% RSLogix 500 project ON DELAY.RSS, saved by version 8.30.00.16 %
PROJECT "UNTITLED"    % processor: MicroLogix 1000 %

PROGRAM FILES
  LAD 2 "MAIN_PROG"  4 rungs
  LAD 3 "START"  9 rungs
  LAD 4 "BUZZER"  7 rungs
  LAD 5 "STI_INT"  1 rungs
  LAD 6, 7, 8, 9, 10, 11, 12, 13, 14, 15, 16: only END

DATA FILES
  O0 OUTPUT  1 elements
  I1 INPUT  2 elements
  S2 STATUS  33 elements
  B3 BINARY  32 elements
  T4 TIMER  40 elements
  C5 COUNTER  32 elements
  R6 CONTROL  16 elements
  N7 INTEGER  105 elements

LADDER 2 "MAIN_PROG"
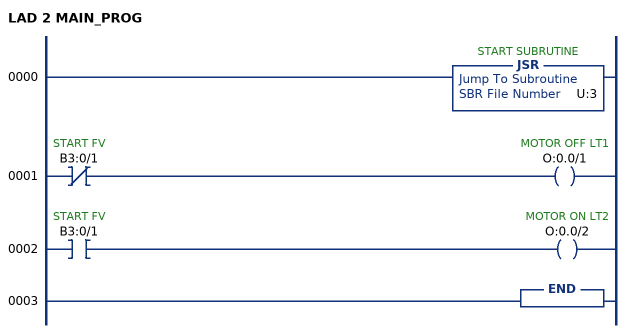
% Rung: 0 %
SOR JSR U:3 EOR
%   U:3  "START SUBRUTINE" %
% Rung: 1 %
SOR XIO B3:0/1 OTE O:0.0/1 EOR
%   B3:0/1  FV  "START" %
%   O:0.0/1  LT1  "MOTOR OFF" %
% Rung: 2 %
SOR XIC B3:0/1 OTE O:0.0/2 EOR
%   B3:0/1  FV  "START" %
%   O:0.0/2  LT2  "MOTOR ON" %
% Rung: 3 %
SOR END EOR

LADDER 3 "START"
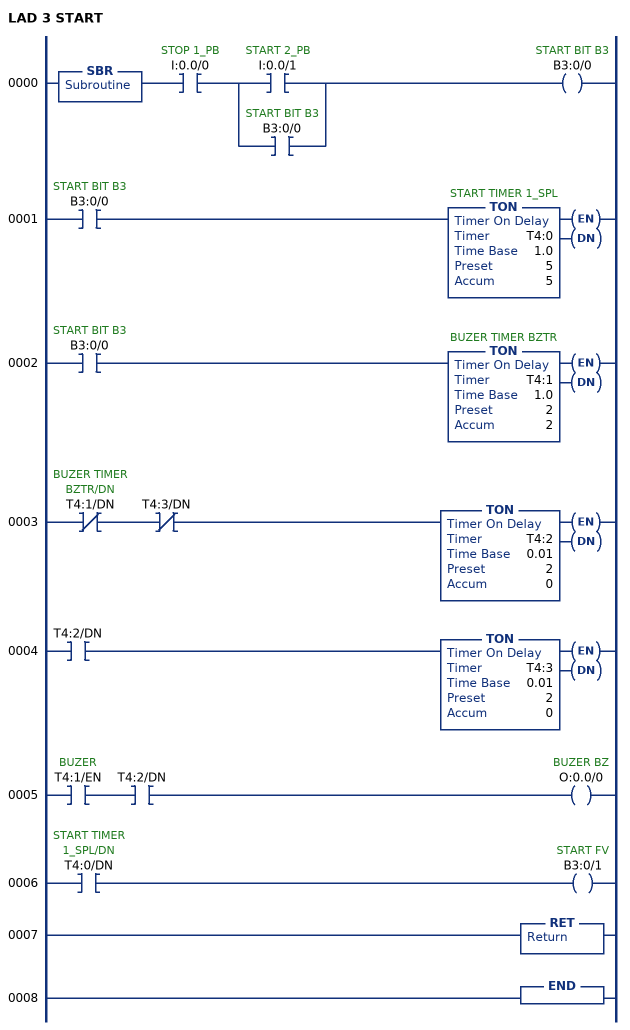
% Rung: 0 %
SOR SBR XIC I:0.0/0 BST XIC I:0.0/1 NXB XIC B3:0/0 BND OTE B3:0/0 EOR
%   I:0.0/0  1_PB  "STOP" %
%   I:0.0/1  2_PB  "START" %
%   B3:0/0  B3  "START BIT" %
% Rung: 1 %
SOR XIC B3:0/0 TON T4:0 1.0 5 5 EOR
%   B3:0/0  B3  "START BIT" %
%   T4:0  1_SPL  "START TIMER" %
% Rung: 2 %
SOR XIC B3:0/0 TON T4:1 1.0 2 2 EOR
%   B3:0/0  B3  "START BIT" %
%   T4:1  BZTR  "BUZER TIMER" %
% Rung: 3 %
SOR XIO T4:1/DN XIO T4:3/DN TON T4:2 0.01 2 0 EOR
%   T4:1  BZTR  "BUZER TIMER" %
% Rung: 4 %
SOR XIC T4:2/DN TON T4:3 0.01 2 0 EOR
% Rung: 5 %
SOR XIC T4:1/EN XIC T4:2/DN OTE O:0.0/0 EOR
%   T4:1/EN  "BUZER" %
%   O:0.0/0  BZ  "BUZER" %
% Rung: 6 %
SOR XIC T4:0/DN OTE B3:0/1 EOR
%   T4:0  1_SPL  "START TIMER" %
%   B3:0/1  FV  "START" %
% Rung: 7 %
SOR RET EOR
% Rung: 8 %
SOR END EOR

LADDER 4 "BUZZER"
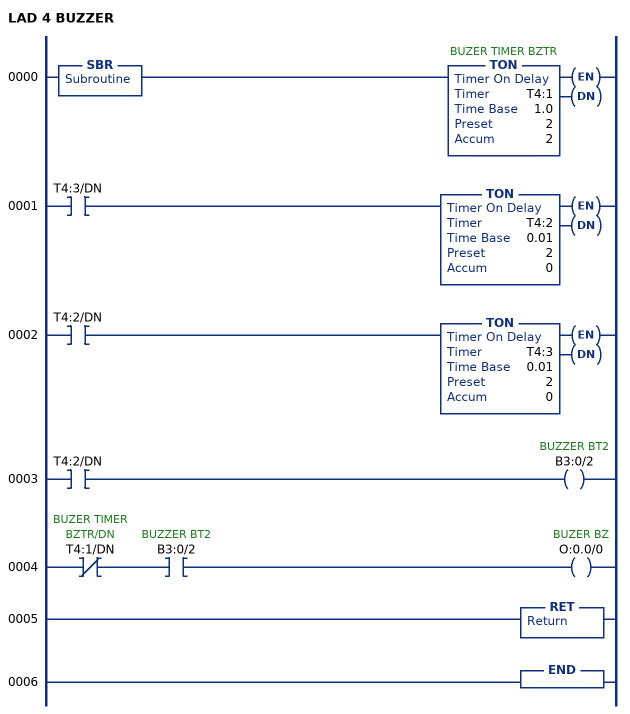
% Rung: 0 %
SOR SBR TON T4:1 1.0 2 2 EOR
%   T4:1  BZTR  "BUZER TIMER" %
% Rung: 1 %
SOR XIC T4:3/DN TON T4:2 0.01 2 0 EOR
% Rung: 2 %
SOR XIC T4:2/DN TON T4:3 0.01 2 0 EOR
% Rung: 3 %
SOR XIC T4:2/DN OTE B3:0/2 EOR
%   B3:0/2  BT2  "BUZZER" %
% Rung: 4 %
SOR XIO T4:1/DN XIC B3:0/2 OTE O:0.0/0 EOR
%   T4:1  BZTR  "BUZER TIMER" %
%   B3:0/2  BT2  "BUZZER" %
%   O:0.0/0  BZ  "BUZER" %
% Rung: 5 %
SOR RET EOR
% Rung: 6 %
SOR END EOR

OTHER DOCUMENTED ADDRESSES
  U:4  "BUZZER SUBRUTINE"

DATA TABLE (non-zero values as saved)
DATA B3
% B3:0 % 0X0003 0X000F 0X0001 0X0002 0X0004 0X0008 0X0009 0X0006 0X000A 0X0005
% B3:10 % 0X0003 0X0005 0X0009 0X000C 0X000A 0X0009 0X0000 0X0000 0X0000 0X0000
DATA T4
% .PRE .ACC %
% T4:0 % 5 5
% T4:1 % 2 2
% T4:2 % 2 0
% T4:3 % 2 0
